(*
SPDX-FileCopyrightText: © 2026 Oleksandr Tiutyk <trofimich@gmail.com>
SPDX-License-Identifier: MIT
License: https://opensource.org/license/mit
*)

(*!
<summary>Condition that is always configured and always evaluates to TRUE.</summary>
*)

{attribute 'no_explicit_call' := 'do not call this function block directly'}
{attribute 'enable_dynamic_creation'}
FUNCTION_BLOCK TrueCondition EXTENDS Condition IMPLEMENTS ITrueCondition, TOF_Core.IConfigurationSerializable
VAR_STAT
	{attribute 'hide'}
	_ClassName : STRING := __POUNAME();
END_VAR

(*!
<summary>Borrows the initialized class name used in diagnostics.</summary>
<description>
Returns initialized metadata storage without allocation. Callers must not modify the returned string.
Derived function blocks must use distinct initialized static storage when overriding this metadata.
</description>
*)
{attribute 'monitoring' := 'call'}
PROPERTY ClassName : REFERENCE TO STRING
GET
ClassName REF= _ClassName;
END_GET
END_PROPERTY

(*!
<summary>Always returns TRUE.</summary>
*)
{attribute 'monitoring' := 'call'}
PROPERTY Configured : BOOL
GET
Configured := TRUE;
END_GET
END_PROPERTY

(*!
<summary>Borrows the compiler-initialized library namespace.</summary>
<description>
Borrows storage from the live internal namespace provider. Reacquire references after application
reinitialization or relocation. Treat the reference as read-only; no ownership or synchronization is provided.
</description>
*)
{attribute 'monitoring' := 'call'}
PROPERTY NamespaceName : REFERENCE TO STRING
GET
NamespaceName REF= CurrentNamespace.Name;
END_GET
END_PROPERTY

(*!
<summary>Always returns TRUE.</summary>
<param name="activity">Unused activity context.</param>
*)
METHOD PROTECTED OnEvaluate : BOOL
VAR_INPUT
	activity : IActivity;
END_VAR
OnEvaluate := TRUE;
END_METHOD

(*!
<summary>Reports the size of this concrete function block instance in bytes.</summary>
<description>
Reports the instance layout rather than dynamic allocations owned by its fields. A derived function block
with a different layout must override this property; the value does not grant disposal rights.
</description>
*)
{attribute 'monitoring' := 'call'}
PROPERTY SelfSize : ULINT
GET
SelfSize := XSIZEOF(THIS^);
END_GET
END_PROPERTY

(*!
<summary>Writes the configuration fields for this object.</summary>
<description>Borrows the writer for this call. A failure invalidates the current output document.</description>
*)
METHOD Serialize
VAR_INPUT
	writer : TOF_Core.IConfigurationWriter;
END_VAR
Workflows.WriteConfigurationHeader(
	writer := writer,
	source := THIS^,
	displayName := Name,
	scope := THIS^
);
END_METHOD

(*!
<summary>Restores this fresh instance from its configuration object.</summary>
<description>
The reader and document node are borrowed for this call. On failure discard the partial instance.
</description>
<param name="reader">Active configuration reader.</param>
<param name="node">Object node to read fields from.</param>
<param name="context">Configuration deserialization context; ignored by this context-free element.</param>
*)
METHOD Deserialize
VAR_INPUT
	reader : TOF_Core.IConfigurationReader;
	node : TOF_Core.CONFIGURATION_NODE;
	context : TOF_Core.IConfigurationDeserializationContext;
END_VAR
Workflows.ReadConfigurationHeader(reader := reader, node := node, target := THIS^, scope := THIS^);
END_METHOD

END_FUNCTION_BLOCK

(* stored: Version 1.1.0.1
   POU TrueCondition: Id {6bc6dfef-1fc1-4a89-87d9-be965cbae9a5}, SpecialFunc None
   Folder Overriden methods: Id {4adee19e-31c9-47ed-8975-c42c758e870a}
   Property ClassName: Id {be399689-ccac-49cf-b5b0-553e97ea68b6}
   Get Get: Id {cf6990c4-9222-443d-be50-67c58aaab94c}
   Property Configured: Id {1cb0bac0-7c56-461e-8a5a-caf7e2db2aae}
   Get Get: Id {99928473-b51e-4e14-93dc-9177537b664f}
   Property NamespaceName: Id {23150ecb-e47e-4e81-8845-52c0606c2451}
   Get Get: Id {24c5d898-0efa-406c-b367-56828e83aa1b}
   Method OnEvaluate: Id {cb24fab5-bc77-4057-929a-28eb3b8af344}
   Property SelfSize: Id {d4cd10d5-9a3b-4938-9776-2a6aa7cc1c92}
   Get Get: Id {7d26d634-58f9-4fdd-8848-6e2e6a5a6bff}
   Method Serialize: Id {5a3787da-0f24-48cf-91bf-959fb2305c3f}
   Method Deserialize: Id {5b73cfce-70fc-443a-b527-6b6b7453e85d} *)
